INTERFACE I_HE_SATT_FilterCombinationCollector


METHOD PUBLIC AddFilterCombination
VAR_INPUT
    fbFilterCombination : REFERENCE TO FB_HE_SATT_FilterCombination;
END_VAR
END_METHOD


METHOD PUBLIC DownselectByCouplingRule
VAR_INPUT
    iFilterCombinationCollector : I_HE_SATT_FilterCombinationCollector;
    iFilterHolderSelector : I_HE_SATT_FilterHolderSelector;
END_VAR
END_METHOD


PROPERTY DownselectStatus : REFERENCE TO ST_HE_SATT_Status
GET
END_GET
END_PROPERTY


METHOD GetCombination : REFERENCE TO FB_HE_SATT_FilterCombination
VAR_INPUT
    nCombinationNumber : DINT;
END_VAR
END_METHOD


PROPERTY NumCombinationsAdded : DINT
GET
END_GET
END_PROPERTY


METHOD PUBLIC Reset
END_METHOD

END_INTERFACE

(* stored: Version 1.1.0.1
   Itf I_HE_SATT_FilterCombinationCollector: Id {d62d89ff-9614-47fb-a95f-4d39cf574fa3}
   Method AddFilterCombination: Id {392deb49-e7c1-42de-a162-b2150e85c96b}
   Method DownselectByCouplingRule: Id {973da3f9-d366-4ead-bda6-e21e8844903c}
   Property DownselectStatus: Id {97279e63-9cd2-42af-8c3b-d22d6c2d5de1}
   Get Get: Id {cf57ad50-186e-46d3-be2c-bd39493d1b73}
   Method GetCombination: Id {4ce62b9d-ae68-40dd-bd58-fb785c38dc50}
   Property NumCombinationsAdded: Id {5f7a125b-9a63-4aa0-852e-b406eaebb5ac}
   Get Get: Id {c4909db4-9c88-4e8b-9e54-c5c601d0e095}
   Method Reset: Id {ba0e24e0-3175-4624-b36e-00ba04724f68} *)
